Staubli VAL3: check_cmt.pgx

public program check_cmt()
  local num sCheck
  local num nEOS
begin

  clearBuffer(sioASCII)

  nEOS = 0
  sCheck = sioSet(sioASCII,nEOS)
  sCheck = sioSet(sioASCII,13)

  if sCheck == 1
    putln("Communication is OK !")
    check_status = true
  elseIf sCheck != 1
    putln("Communication error !")
    check_status = false
  endIf

end
